Yaskawa INFORM job: R1_W53-A1(90,180)R2.JBI

/JOB
//NAME R1_W53-A1(90,180)R2
///FOLDERNAME KRIS-SCIANA
//POS
///NPOS 56,56,0,2,0,0
///TOOL 0
///POSTYPE PULSE
///PULSE
C00000=29586,64241,-25483,43781,98921,43724
C00001=57127,101638,10899,56682,107332,38251
C00002=57127,76182,10095,53684,99903,33351
C00003=68868,95750,33777,40131,101998,35545
C00004=80579,136048,88691,13195,105824,34209
C00005=80579,135466,89528,13135,105030,34121
C00006=80773,138592,94773,13031,103420,34013
C00007=80579,135466,89528,13135,105030,34121
C00008=80098,138136,91616,11040,112385,45139
C00009=80392,131132,88850,2537,121882,58675
C00010=80276,129363,86425,2517,122469,58643
C00011=80392,131132,88850,2537,121882,58675
C00012=78176,133439,87120,21461,107379,43183
C00013=80582,134264,97775,32660,78294,14244
C00014=80553,132262,95759,32645,78486,14287
C00015=83645,119224,78721,23719,77537,14384
C00016=83470,121059,81194,23821,77054,14221
C00017=80306,137503,105397,33060,75839,13403
C00018=79806,133260,94028,32682,80109,14466
C00019=76874,109703,51513,11024,106473,-11901
C00020=80591,100267,38822,2686,105144,-12380
C00021=80592,98128,39662,2663,103530,-12415
C00022=78991,102203,46514,6213,103180,-12291
C00023=80323,95098,37876,2698,103081,-12510
C00024=80415,96751,38231,2692,103708,-12467
C00025=79562,99039,43342,-2010,99419,-12297
C00026=80580,97640,39756,-2642,100727,-11961
C00027=80580,99717,38880,-2660,102332,-11996
C00028=78782,132344,81667,13923,102302,-75965
C00029=80359,118001,67121,13069,108526,-74927
C00030=75015,121502,76672,18597,108324,-76052
C00031=72170,117106,73613,18379,108585,-77056
C00032=72430,123841,78142,18479,109171,-76865
C00033=74362,68166,3081,6175,104558,-36694
C00034=69157,63041,7727,10776,93973,-38093
C00035=69752,61654,6114,10607,94178,-37894
C00036=73709,53321,-3394,9465,95292,-36609
C00037=75219,53872,-3292,7232,98435,-36398
C00038=74402,58837,-4462,7542,101743,-36441
C00039=77887,55118,-12218,6694,104332,-35282
C00040=73093,73480,10032,23382,107480,-22737
C00041=73093,73480,10032,23382,107480,-48018
C00042=75077,67955,12819,31918,102727,-41123
C00043=72358,72933,20789,32098,101649,-42430
C00044=69710,68999,13649,32933,104577,-42537
C00045=73972,81494,17525,17998,114452,-43214
C00046=73978,81364,17362,17976,114428,-384
C00047=76924,75829,15003,17496,112550,309
C00048=74228,52611,-5361,20593,98975,-1808
C00049=77356,54576,-3191,19708,98006,-990
C00050=76013,58955,1854,22690,99776,-4336
C00051=73409,62701,9144,33997,102367,-2022
C00052=68667,63426,3503,35642,107245,-2197
C00053=76429,128622,61528,15029,112853,-75461
C00054=76429,128622,61528,15029,59041,-75461
C00055=49009,130387,53171,15969,61359,76811
BC00000=15470,555342,1075171
BC00001=15470,482644,1075171
BC00002=15470,482644,1075171
BC00003=15470,482644,1075171
BC00004=15469,482644,1075175
BC00005=15999,482682,1075175
BC00006=15999,482682,1075175
BC00007=15999,482682,1075175
BC00008=17464,460994,1075175
BC00009=19492,430987,1075175
BC00010=19492,430987,1075175
BC00011=19492,430987,1075175
BC00012=20512,473832,1075175
BC00013=21980,535468,1075175
BC00014=21994,538910,1075175
BC00015=21994,538910,1075175
BC00016=21994,538910,1075175
BC00017=21994,538910,1075175
BC00018=21994,538910,1075175
BC00019=871,485532,1075175
BC00020=871,485532,1075175
BC00021=1360,481393,1075175
BC00022=1421,480878,1075175
BC00023=1555,479738,1075175
BC00024=1555,479738,1075175
BC00025=26602,479127,1075175
BC00026=28340,480604,1075175
BC00027=27012,484692,1075175
BC00028=26690,484644,1075175
BC00029=26690,468991,1075175
BC00030=26690,468991,1075175
BC00031=26690,468991,1075175
BC00032=26690,468991,1075175
BC00033=26690,468991,1075175
BC00034=26690,468991,1075175
BC00035=26690,468991,1075175
BC00036=26690,468991,1075175
BC00037=26690,468991,1075175
BC00038=26690,468991,1075175
BC00039=26690,468991,1075175
BC00040=26690,468991,1075175
BC00041=26690,468991,1075175
BC00042=26690,468991,1075175
BC00043=26690,468992,1075173
BC00044=26690,468992,1075173
BC00045=26690,468992,1075173
BC00046=26690,468992,1075173
BC00047=26690,468992,1075173
BC00048=26690,468992,1075173
BC00049=26690,468992,1075173
BC00050=26690,468992,1075173
BC00051=26690,468992,1075173
BC00052=26690,468992,1075173
BC00053=26690,484644,1075175
BC00054=26690,525723,1075175
BC00055=26690,531768,1075175
///POSTYPE BASE
///RECTAN
///RCONF 0,0,0,0,1,0,0,0,0,0,0,0,0,0,0,0,0,0,0,0,0,0,0,0
P00006=2.006,1.622,-0.565,0.0000,0.0000,0.0000
P00022=2.006,1.622,-0.565,0.0000,0.0000,0.0000
//INST
///DATE 2024/11/08 13:14
///ATTR SC,RW
///GROUP1 RB1,BS1
NOP
'r2_W53-A1(90,180)
'Path S1056
SFTOF
MOVJ C00000 BC00000 VJ=20.00
MOVJ C00001 BC00001 VJ=10.00
MOVJ C00002 BC00002 VJ=20.00
MOVJ C00003 BC00003 VJ=20.00
MOVL C00004 BC00004 V=100.0
MOVL C00005 BC00005 V=60.0
REFP 3 C00006 BC00006
CALL JOB:SEARCH-R1
SET P022 P006
SFTON P022
MOVL C00007 BC00007 V=60.0
MOVL C00008 BC00008 V=60.0
MOVL C00009 BC00009 V=100.0
REFP 3 C00010 BC00010
CALL JOB:SEARCH-R1
SET P022 P006
SFTON P022
MOVL C00011 BC00011 V=100.0
MOVL C00012 BC00012 V=60.0
MOVL C00013 BC00013 V=100.0
MOVL C00014 BC00014 V=60.0
MOVL C00015 BC00015 V=60.0
REFP 3 C00016 BC00016
CALL JOB:SEARCH-R1
SET P022 P006
SFTON P022
MOVL C00017 BC00017 V=60.0
MOVL C00018 BC00018 V=100.0
'Path W1057
SFTOF
SFTON P022
MOVJ C00019 BC00019 VJ=20.00
MOVJ C00020 BC00020 VJ=20.00 PL=0
CALL JOB:COFNIJ_DRUT
MOVL C00021 BC00021 V=100.0
MOVL C00022 BC00022 V=100.0 PL=0
REFP 1 C00023 BC00023
REFP 2 C00024 BC00024
MACRO1 MJ#(0) ARGF7
ARCON
MOVL C00025 BC00025 V=10.8
ARCOF
MOVL C00026 BC00026 V=100.0
MOVL C00027 BC00027 V=166.7
SFTOF
SFTON P022
'COMMENT
MOVJ C00028 BC00028 VJ=20.00
MOVL C00029 BC00029 V=100.0 PL=0
MACRO1 MJ#(0) ARGF6
ARCON
MOVL C00030 BC00030 V=8.3
MOVL C00031 BC00031 V=8.3
ARCOF
MOVL C00032 BC00032 V=100.0
MOVL C00033 BC00033 V=100.0
COMM MACRO1 MJ#(0) ARGF6
COMM MOVL C00034 BC00034 V=83.3
COMM ARCON
COMM MOVL C00035 BC00035 V=10.0
COMM MOVL C00036 BC00036 V=10.0
COMM MOVL C00037 BC00037 V=10.0
COMM ARCOF
COMM MOVJ C00038 BC00038 VJ=10.00
MOVJ C00039 BC00039 VJ=10.00
MOVJ C00040 BC00040 VJ=10.00
MOVJ C00041 BC00041 VJ=10.00
MACRO1 MJ#(0) ARGF7
MOVJ C00042 BC00042 VJ=10.00
ARCON
MOVL C00043 BC00043 V=8.3
ARCOF
MOVJ C00044 BC00044 VJ=10.00
MOVJ C00045 BC00045 VJ=10.00
MOVJ C00046 BC00046 VJ=10.00
MOVJ C00047 BC00047 VJ=10.00
MOVJ C00048 BC00048 VJ=10.00
ARCON
MOVL C00049 BC00049 V=10.0
MOVL C00050 BC00050 V=10.0
MOVL C00051 BC00051 V=10.0
ARCOF
MOVJ C00052 BC00052 VJ=10.00
MOVJ C00053 BC00053 VJ=40.00
MOVJ C00054 BC00054 VJ=100.00
SFTOF
MOVJ C00055 BC00055 VJ=100.00
END
